SYSTEM BasicIcaruIo (* System Configuration *)
  (* Standard: 61499-1 *)
  (* Version 0.4, 2009-03-05, JHC, Holobloc Inc., Deleted Application. *)
  (* Version 0.3, 2003-12-05, JHC, Rockwell Automation, Renamed from NEWSYSTEM. *)
  (* Version 0.2, 2002-11-05, JHC, Rockwell Automation, Fixed missing (empty) FBD in Application. *)
  (* Version 0.1, 2002-01-17, JHC, Rockwell Automation, Minor cleanup *)
  (* Version 0.0, 2000-05-27, JHC, Rockwell Automation *)
  DEVICE ICARU4442 : RMT_DEV(MGR_ID := "localhost:61494")
    RESOURCE RESM : EMB_RES
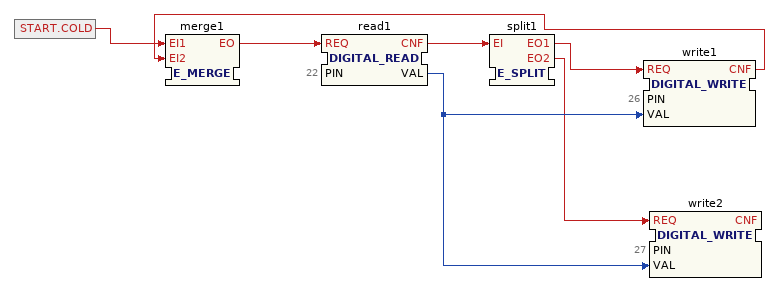
      FBS
        read1 : DIGITAL_READ(PIN := 22);
        write1 : DIGITAL_WRITE(PIN := 26);
        merge1 : E_MERGE;
        split1 : E_SPLIT;
        write2 : DIGITAL_WRITE(PIN := 27);
      END_FBS
      EVENT_CONNECTIONS
        START.COLD TO merge1.EI1;
        merge1.EO TO read1.REQ;
        write1.CNF TO merge1.EI2;
        read1.CNF TO split1.EI;
        split1.EO1 TO write1.REQ;
        split1.EO2 TO write2.REQ;
      END_CONNECTIONS
      DATA_CONNECTIONS
        read1.VAL TO write1.VAL;
        read1.VAL TO write2.VAL;
      END_CONNECTIONS
    END_RESOURCE
  END_DEVICE
END_SYSTEM
